TYPE ST_Space :
STRUCT
	bIsOccupied		: BOOL;
	sPartID			: STRING(23);
END_STRUCT
END_TYPE

(* stored: Version 1.1.0.1
   DUT ST_Space: Id {7525ade0-a898-4674-8c67-32f602dcdcda} *)
